Universal Robots PolyScope program: Ejercicio_3.urp

Program Ejercicio_3 (installation=default directory=/home/ur/ursim-current/programs/Ejercicio_3 createdIn=5.7.0.90932 lastSavedIn=5.7.0.90932 robotSerialNumber=20195599999)
Calibrated DH parameters: a=[0, -0.425, -0.3922, 0, 0, 0]; d=[0.1625, 0, 0, 0.1333, 0.0997, 0.0996]; alpha=[1.570796, 0, 0, 1.570796, -1.570796, 0]; deltaTheta=[0, 0, 0, 0, 0, 0]
Robot Program (runOnlyOnce=true)
  Script file /home/ur/ursim-current/programs/Ejercicio_3/Ejercicio_3.script
    |      # Preparar instalacion
    |       set_gravity([0,0,9.8])
    |       set_payload_mass(3)
    | 
    |      # Configuración herramientas
    |       t_desbarb=p[0.05, 0.025, 0.175,0,0,1.57] # herramienta desbarbado
    |       t_pulido=p[-0.05, 0.025, 0.175,0,0,1.57] # herramienta pulido
    | 
    |       # Variables
    |       varx = 0
    |       vary = 0
    |       n_filas = 2.0
    |       n_columnas = 2.0
    |       d_filas = 0.02
    |       d_columnas = 0.02
    | 
    |       #rutina de desbarbado
    |       def desbarbado(varx, vary, n_filas, n_columnas, d_filas, d_columnas):
    |        i=1
    |        j=1
    |        set_tcp(t_desbarb)
    |        set_digital_out(0,True)
    |        while i <= n_columnas:
    |         while  j <= n_filas:
    |          pose_pre = p[0.5+varx,-0.150+vary,0.05,0,3.1416,0]
    |          pose_desb = p[0.5+varx,-0.150+vary,0,0,3.1416,0]
    |          movej(pose_pre,1.5,1) #acercamiento
    |          movel(pose_desb,1.5,1) #punto desbarbado
    |          sleep(2.5)
    |          movej(pose_pre,1.5,1) #salida
    |          textmsg("Desbarbado en fila "+to_str(j)+" columna "+to_str(i)+" finalizado")
    |          varx=varx+d_filas
    |          j=j+1
    |         end
    |        varx=0
    |        j=1
    |        vary=vary+d_columnas
    |        i=i+1
    |       end
    |       set_digital_out(0,False)
    |       end
    | 
    |     #rutina de pulido
    |       def pulido(varx, vary, n_filas, n_columnas, d_filas, d_columnas):
    |       i=1
    |       j=1
    |        set_tcp(t_pulido)
    |        set_digital_out(1,True)
    |        while i <= n_columnas:
    |         while  j <= n_filas:
    |          pose_pre = p[0.5+varx,-0.150+vary,0.05,0,3.1416,0]
    |          pose_desb = p[0.5+varx,-0.150+vary,0,0,3.1416,0]
    |          movej(pose_pre,1.5,1) #acercamiento
    |          movel(pose_desb,1.5,1) #punto desbarbado
    |          sleep(1)
    |          movej(pose_pre,1.5,1) #salida
    |          textmsg("Pulido en fila "+to_str(j)+" columna "+to_str(i)+" finalizado")
    |          varx=varx+d_filas
    |          j=j+1
    |         end
    |        varx=0
    |        j=1
    |        vary=vary+d_columnas
    |        i=i+1
    |       end
    |       set_digital_out(0,False)
    |       end
    | 
    |       #Programa
    |       set_tcp(t_desbarb)
    |       popup("Iniciando programa desbarbado/pulido rejillas",title="Info",warning=False,blocking=True)
    |       textmsg("Iniciando programa")
    |       safe_pose = [0,-0.78,-1.57,-2.35,1.57,0]
    |       movej(safe_pose,1.5,1)
    |       desbarbado (varx, vary, n_filas, n_columnas, d_filas, d_columnas)
    |       movej(safe_pose,1.5,1)
    |       pulido (varx, vary, n_filas, n_columnas, d_filas, d_columnas)
    |       movej(safe_pose,1.5,1)
    |       textmsg("Programa finalizado")
    |       popup("Programa desbarbado/pulido rejillas finalizado",title="Info",warning=False,blocking=True)
